{attribute 'qualified_only'}
{attribute 'strict'}
{attribute 'to_string'}
TYPE DUT_Command_CoordinateType :
(
	Literal := 0,
	Variable := 1
);
END_TYPE

(* stored: Version 1.1.0.1
   EnumerationTextList DUT_Command_CoordinateType: Id {208151aa-6cb4-4b6a-b40b-958da433a410} *)
